// TIA Portal V18 export
FUNCTION "AHU_Main" : Void   // FC100, FBD
{ S7_Optimized_Access := 'TRUE' }
VERSION : 0.1
// stored: AutoNumber false, IsIECCheckEnabled false, SetENOAutomatically false, UDAEnableTagReadback false
   VAR_INPUT
      iUnitID : Int;   // 1=AHUFood, 2=AHUNonFood
   END_VAR
   VAR_TEMP
      FA_temp : Real;
   END_VAR
BEGIN

REGION Network 1 (SCL): Actual Room (salles area temp)
   // 0=PLC_IO, 1=LoraAvg, 2=MSensor,3 =PLC
   CASE "AHUAI".AI.cRoomTempSelect[#iUnitID] OF
       0:  // 
           "AHUAI".AI.rRoomAirTemp_Actual[#iUnitID] := "AHUAI".AI.rRoomAirTemp_PLC_AI[#iUnitID];
       1:  // 
           "AHUAI".AI.rRoomAirTemp_Actual[#iUnitID] := "AHUAI".AI.rRoomAirTemp_LoraAvg[#iUnitID];
       2: // 
           "AHUAI".AI.rRoomAirTemp_Actual[#iUnitID] := "AHUAI".AI.rRoomAirTemp_MSensor[#iUnitID];
       ELSE
           "AHUAI".AI.rRoomAirTemp_Actual[#iUnitID] := "AHUAI".AI.rRoomAirTemp_PLC_AI[#iUnitID];
   END_CASE;
END_REGION

REGION Network 2
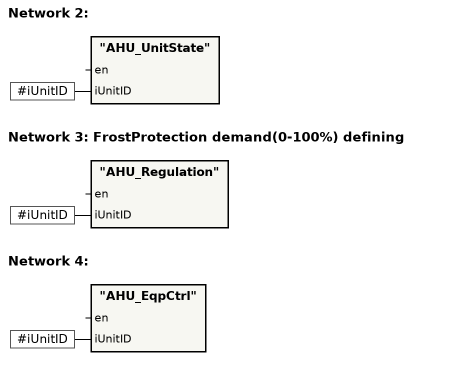
   "AHU_UnitState"(iUnitID := #iUnitID);
END_REGION

REGION Network 3: FrostProtection demand(0-100%) defining
   "AHU_Regulation"(iUnitID := #iUnitID);
END_REGION

REGION Network 4
   "AHU_EqpCtrl"(iUnitID := #iUnitID);
END_REGION
END_FUNCTION
